// TIA Portal V19 export
DATA_BLOCK "DI MAPING"   // DB1
{ S7_Optimized_Access := 'TRUE' }
// stored: MemoryReserve 100
   VAR
      "EMG STOP-1" : Bool;
      "EMG STOP-2" : Bool;
      "HOOTER RESET-1" : Bool;
      "HOOTER RESET-2" : Bool;
      "AIR PRESSURE SWITCH" : Bool;
      "PHASE FAIL" : Bool;
      "MFG VESSEL MOTOR TRIP" : Bool;
      "PREMIXING VESSEL MOTOR TRIP" : Bool;
      "STORAGE VESSEL-1 MOTOR TRIP" : Bool;
      "STORAGE VESSEL-2 MOTOR TRIP" : Bool;
      "INLINE HOMOGENIZER-1 TRIP" : Bool;
      "FILTER PRESS MOTOR TRIP" : Bool;
      "INLINE HOMOGENIZER-2 TRIP" : Bool;
      "MFG LOBE PUMP TRIP" : Bool;
      "STORAGE VESSEL-1 LOBE PUMP TRIP" : Bool;
      "STORAGE VESSEL-2 LOBE PUMP TRIP" : Bool;
      "SUGAR VESSEL MOTOR TRIP" : Bool;
      "BASKET FILTER MOTOR TRIP" : Bool;
      "VACUUME PUMP-1 TRIP" : Bool;
      "VACUUME PUMP-2 TRIP" : Bool;
      "CIP FORWARD PUMP TRIP" : Bool;
      "CIP REVERSE PUMP TRIP" : Bool;
      "LEVEL SWITCH LOW-ALKALI" : Bool;
      "LEVEL SWITCH HIGH-ALKALI" : Bool;
      "LEVEL SWITCH LOW-ACID" : Bool;
      "LEVEL SWITCH HIGH-ACID" : Bool;
      "FLOW SWITCH- MFG" : Bool;
      "FLOW SWITCH- PREMIXING" : Bool;
      "FLOW SWITCH- STORAGE VESSEL-1" : Bool;
      "FLOW SWITCH- STORAGE VESSEL-2" : Bool;
      "FLOW SWITCH- SUGAR VESSEL" : Bool;
      "FLOW SWITCH- HMOGENIZER-1" : Bool;
      "FLOW SWITCH- HMOGENIZER-2" : Bool;
      "LEVEL FLOW SWITCH-1" : Bool;
      "LEVEL FLOW SWITCH-2" : Bool;
      "DI SPARE_1" : Bool;
      "DI SPARE_2" : Bool;
      "DI SPARE_3" : Bool;
      "DI SPARE_4" : Bool;
      "DI SPARE_5" : Bool;
   END_VAR
BEGIN
END_DATA_BLOCK
